(* IEC 61131-3 sources: crb-codesys/retrieval/output/codesys_repo/PID_controller/Models, 3 files *)

(* ---- HeatExchanger.st ---- *)
// AJ Jaworowski 2015-02-22
// Following the recipe by  Peter Nachtwey
// http://www.controlguru.com/wp/p80.html
FUNCTION_BLOCK HeatExchanger
VAR_INPUT
	Kp: REAL; //System gain
	Tp: REAL; //Process time
	CO: REAL; //Output from controller
	Dead_t: REAL; //The time before the system responds to the disturbance
	C: REAL; //Initial steady state value
	Sample_time: TIME;
END_VAR
VAR_OUTPUT
	PV: REAL; //Process value at t1
END_VAR
VAR
	now: TIME;
	lastTime: TIME;
	lastPV:REAL := 140;
	A: REAL;
	B: REAL;
	delta_t: REAL;
END_VAR
VAR CONSTANT
	millis: REAL := 1000;
END_VAR

now := TIME();
IF ((now - lastTime) > Sample_time) THEN
	delta_t := TIME_TO_REAL(Sample_time)/millis;
	A := EXP(-delta_t/Tp);
	B := 1 - A;
	C := 2;

	//PV := A * lastPV + B * Kp * CO + C;
	PV := 0.987 * lastPV - 0.00679 * CO + C;
	lastPV := PV;

	lastTime := now;
END_IF

(* ---- HeatExchanger2.st ---- *)
// AJ Jaworowski 2015-02-23
// Following the presentation on
// http://openenergymonitor.org/emon/node/2999
FUNCTION_BLOCK HeatExchanger2
VAR_INPUT
	Heat_In:		REAL;		//In principle a radiator in the room [W]
	U:				REAL;		//Thermal conductance [W/K]
	TC:				REAL;		//Thermal capacity [J/K], commonly cv, specific heat capacity [J/kgK]
								//we use a smaller value than in reality, so that we can see changes
								//during a life-time...
	Temp_In:		REAL;		//Start temperature in the room [K]
	Temp_Out:		REAL;		//Outside temperature [K]
	Sample_time:	TIME;
END_VAR
VAR_OUTPUT
	Temp:			REAL;		//The resulting room temperature
END_VAR
VAR
	now: TIME;
	lastTime: TIME := T#0s;
	delta_t: REAL;
	heat_flow: REAL;
	lastTemp: REAL;
END_VAR
VAR CONSTANT
	millis: REAL := 1000;
END_VAR

now := TIME();
IF ((now - lastTime) > Sample_time) THEN
	delta_t := TIME_TO_REAL(Sample_time)/millis;

	//First calculate net heat
	//Heat_In is our heat source
	//Second term is heat flow depending on temperature difference
	//Obs: At start, set lastTime to start temp Temp_In
	IF lastTime = T#0S THEN
		lastTemp := Temp_In;
	END_IF
	heat_flow := Heat_In - U * (lastTemp - Temp_Out);

	//Second: calculate temperature change due to heat_flow
	Temp := lastTemp + heat_flow * delta_t / TC;

	//Update variables for next iteration
	lastTemp := Temp;
	lastTime := now;
END_IF;

(* ---- Tank.st ---- *)
//A.J. Jaworowski 2015-02-20
//Simulering av en tank med RedBull
FUNCTION_BLOCK Tank
VAR_INPUT
	Process_In: REAL;  //Flöde in per sekund, testa vad som händer on du matar in 100
					   //Därefter ska regulatorns OUT in i denna ingång.
	Process_Out: REAL; //Flöde ut per sekund, typ 90
					   //Effekten blir att tanken fylls med 10 per sekund
					   //Full efter ca 1 minut - testa
	SampleTime: TIME;  //Uppdateringstid, typ 100ms
	Lower_limit: REAL; //Tankens lägsta nivå, typ 0
	Upper_limit: REAL; //Tankens max nivå, kanske 500
END_VAR
VAR_OUTPUT
	Level: REAL; //Nivån i tanken
END_VAR
VAR
	now: TIME;
	lastTime: TIME;
	proc_sum_in: REAL := 0;
	proc_sum_out: REAL := 0;
	temp: REAL;
	millis: UINT := 1000;
	proc_out: REAL;
END_VAR

now := TIME();
IF ((now - lastTime) > SampleTime) THEN
	Level := Level +  TIME_TO_REAL(SampleTime)/millis * (Process_In - Process_Out);
	IF Level < Lower_limit THEN
		Level := Lower_limit;
	ELSIF Level > Upper_limit THEN
		Level := Upper_limit;
	END_IF;
	lastTime := now;
END_IF;
